function_block FB_Syntax_ConditionalCompile  
var  
    nValue : int;  
{IF defined(pou: FB_Syntax_ConditionalCompile)}  
    bFeature : bool;  
{ELSE}
    nLegacy : int;  
{END_IF}  
end_var

{IF defined(pou: FB_Syntax_ConditionalCompile)}  
nValue := 1;
{ELSE}  
nValue := 2;
{END_IF}

END_FUNCTION_BLOCK

(* stored: Version 1.1.0.1, ProductVersion 3.1.4024.16
   POU FB_Syntax_ConditionalCompile: Id {9b4230a4-288c-47e8-b242-cf02e486d584}, SpecialFunc None *)
